(* PLC project input_chain_control, Dassault Systèmes ControlBuild 2024x *)
(* stored: creationDateTime 2023-10-03T11:13:58-01:00 *)

FUNCTION_BLOCK tri_chain.input_chain_control
  VAR_INPUT
    globalRunning : BOOL := false;
    localRunning : BOOL := false;
    startSensor : BOOL := false;
    endSensor : BOOL := false;
    captureEnabled : BOOL := false;
  END_VAR
  VAR_OUTPUT
    movement : BOOL := false;
    captureRequest : BOOL := false;
    captureFinished : BOOL := false;
  END_VAR

INITIAL_STEP 10:
  COMPUTE_FUNCTION_BLOCKS(S);
END_STEP
TRANSITION FROM 10 TO 11
  := startSensor AND NOT endSensor AND globalRunning;
END_TRANSITION
STEP 11:
  11_INLINE1(N);
END_STEP
ACTION 11_INLINE1:
  movement;
END_ACTION
TRANSITION FROM 11 TO 12
  := endSensor;
END_TRANSITION
STEP 12:
END_STEP
TRANSITION FROM 12 TO 13
  := localRunning;
END_TRANSITION
STEP 13:
  13_INLINE2(N);
END_STEP
ACTION 13_INLINE2:
  captureRequest;
END_ACTION
TRANSITION FROM 13 TO 14
  := captureEnabled;
END_TRANSITION
STEP 14:
  14_INLINE3(N);
END_STEP
ACTION 14_INLINE3:
  movement;
END_ACTION
TRANSITION FROM 14 TO 15
  := NOT endSensor;
END_TRANSITION
STEP 15:
  15_INLINE4(N);
END_STEP
ACTION 15_INLINE4:
  captureFinished;
END_ACTION
TRANSITION FROM 15 TO 10
  := NOT captureEnabled;
END_TRANSITION
ACTION COMPUTE_FUNCTION_BLOCKS:  (* blocks drawn on the SFC sheet *)
  G1:
END_ACTION
END_FUNCTION_BLOCK
